FUNCTION_BLOCK FB_ServerWait
(*Listioning and accecpt connect for remote*)
VAR_INPUT
	bEnable : BOOL;
	sLocalHost : STRING(15) := '192.168.1.100';//'192.168.1.245';'192.168.137.74'
	nLocalPort : UINT := 4999;

END_VAR
VAR_OUTPUT
	hSocket : T_HSOCKET;
	bBusy: BOOL;
	bError: BOOL;
	nErrID : UDINT;
END_VAR
VAR
	fblisten :FB_SocketListen := (sSrvNetID := '');	
	fbAccept : FB_SocketAccept;
	fbClose : FB_SocketClose;
	fbReconncetTon: TON:=(PT := GVL.Reconnect_time);
	fbAcceptTon: TON:=(PT := GVL.AcceptTime);
		
	hListener : T_HSOCKET;	
	
	bListening : BOOL;
	bAccepting : BOOL;
	
	step : UINT := 0;
	
END_VAR

CASE step OF
	0:(*Init*)
		IF bEnable THEN
			fbReconncetTon(IN := FALSE);
			fblisten(bExecute := FALSE);
			step := 10;
			bBusy:= TRUE;
			nErrID := 0;
			bError := FALSE;
		END_IF
	10:(*Start listenin*)
		fbReconncetTon(IN := TRUE, PT := GVL.Reconnect_time);
		IF fbReconncetTon.Q THEN
			fblisten(sLocalHost := sLocalHost,
			nLocalPort := nLocalPort,
			bExecute := TRUE,
			tTimeout := GVL.ListenTime);
			step := 15;	
		END_IF
						
	15:(*Listening*)
		fbListen(bExecute := FALSE);
		bListening := TRUE;
		IF NOT fbListen.bBusy THEN
			IF NOT fbListen.bError THEN
				hListener := fbListen.hListener; 
				
				step := 20;
				(*prepare for accept*)
				fbAcceptTon(IN:=FALSE);
				fbAccept(bExecute := FALSE);
			ELSE
				bError := TRUE;				
				nErrID := fbListen.nErrId;
				step := 100;
			END_IF
		END_IF
	20:(*start to accept*)	
		bListening := FALSE;
		fbAcceptTon(IN := TRUE,PT := GVL.AcceptTime);
		IF fbAcceptTon.Q THEN
			fbAcceptTon(IN :=FALSE);
			fbAccept(hListener := hListener, bExecute := TRUE);
			step := 25;
		END_IF
	25: (* Accepting*)
		fbAccept(bExecute := FALSE);
		bAccepting := TRUE;
		IF NOT fbAccept.bBusy THEN
			IF NOT fbAccept.bError THEN
				(*check if there is connection be accepted*)
				IF fbAccept.bAccepted THEN
					hSocket := fbAccept.hSocket;
					bBusy := FALSE;
					step := 40;
				ELSE
					step := 20;
				END_IF	
							
			ELSE
				bError := TRUE;
				nErrID := fbAccept.nErrId;
				step := 100;	
			END_IF
		END_IF
		
	40:(*wait for new connect*)
		bBusy := TRUE;
		step:= 20;
	100:(*deal with error*)
		step := 0;
		
		
END_CASE

END_FUNCTION_BLOCK

(* stored: Version 1.1.0.1, ProductVersion 3.1.4022.12
   POU FB_ServerWait: Id {ed199503-4219-4dd1-8488-4a55422b2c84}, SpecialFunc None *)
